// SIMATIC S7-200 project (STEP 7-Micro/WIN), CPU 224 REL 02.01

SYMBOL_TABLE USER1
低压泵延时启动高压        T120
慢驱制动泵启动延时        T110
低压压力正常延时         T109
高压泵工作延时          T108
十分钟停高压泵          T105
运行信号延时           T104
延时停低压泵           T103
再次启高压后停高压        T102
巡检议超温延时          T101
主电机加热            Q5.5
机旁控制指示           Q4.7
机旁反转慢驱指示         Q4.6
机旁正转指示           Q4.5
机旁润滑指示           Q4.4
稀油站出油口温度高        Q4.2
稀油站油位异常          Q4.1
稀油站过滤器故障         Q4.0
稀油站高压油压低         Q3.3
稀油站低压油压低         Q3.2
润滑站油位异常          Q3.1
润滑站油压异常          Q3.0
停止干油泵            Q2.6
系统启动             Q2.5
油站备妥指示           Q2.4
干油泵工作            Q2.3
综合故障输出           Q2.2
停主机信号            Q2.1
油站备妥输出           Q2.0
慢驱油泵工作           Q1.0
慢驱反转             Q0.7
慢驱正转             Q0.6
六泵工作             Q0.5
五泵工作             Q0.4
四号低压泵工作          Q0.3
三号低压泵工作          Q0.2
二泵高压泵工作          Q0.1
一泵高压泵工作          Q0.0
主机停后停干油泵中继       M10.4
慢驱主电机启动前保护       M10.1
慢驱主电机启动后保护       M10.0
停主机中继            M3.3
四号低压泵备用          M3.2
三号低压泵备用          M3.1
总起条件不满足          M3.0
五号润滑泵备用          M2.6
六号润滑泵备用          M2.5
首选手动控制           M2.3
首选自动控制           M2.2
首选机旁控制           M2.1
总起条件             M2.0
急停后再次启高压         M1.5
超温故障停车           M1.6
主机运行记忆           M1.4
主机运行前停车          M1.3     // 主机运行前的停车
高压泵工作            M1.0
启动高压泵            M0.7
低压泵工作            M0.5
手动控制中继           M0.1
内部零电压保护          M0.0
润滑站油温高           I5.7
润滑站油位低           I5.6
润滑站油位高           I5.5
机旁反转慢驱           I5.4
机旁正转慢驱           I5.3
机旁起停润滑           I5.2
机旁启动低压泵          I5.1
机旁起停高压泵          I5.0
润滑油压低            I4.7
润滑压力正常           I4.6
润滑站油压高           I4.5
主机运行             I4.4
低压高              I4.3
稀油站低压低           I4.2
油箱温度低            I4.1
油箱油温高            I4.0
油箱油位低            I3.7
油箱油位高            I3.6
出口油温低            I3.5
出口油温高            I3.4
高低压油站过滤器故障       I3.3
二号高压泵压力低         I3.2
一号高压泵压力低         I3.1
巡检仪超温输入          I3.0
主辅离合器            I2.7     // 开主机为常开
慢驱保护             I2.6
六号泵保护            I2.5
五号泵保护            I2.4
四号泵保护            I2.3
三号泵保护            I2.2
二号泵保护            I2.1
一号泵保护            I2.0
油流控制             I1.5
润滑泵起停            I1.4
低压泵起停            I1.3
高压泵起停            I1.2
润滑泵选择            I1.1
主电机加热温度上限        I0.7
低压泵选择            I1.0
手动加热             I0.6
反转慢驱             I0.5
正转慢驱             I0.4
自动控制             I0.3
机旁控制             I0.2
总起动              I0.1
急停               I0.0     // 主机、机旁、本柜
END_SYMBOL_TABLE

ORGANIZATION_BLOCK 攀枝花紫东钛综合柜程序:OB1
TITLE=【攀枝花矿业公司的空气扫风磨机的自动化控制系统】
// 系统启动前，会检查多项条件，例如油流控制传感器必须正常、主机运行传感器必须未运行、慢驱主电机启动后保护必须未触发，只有这些条件都满足时，总起条件才会置位，允许系统进入运行状态。
// 运行时，系统根据选定的模式和传感器反馈，驱动多个设备。例如，在自动模式下，若油流控制传感器正常且油箱油位低传感器未触发，系统会根据低压泵选择开关的状态，启动三号低压泵工作或四号低压泵工作，但前提是三号泵保护传感器和四号泵保护传感器必须正常，否则泵不会运行。类似地，五号润滑泵工作和六号润滑泵工作的启动需要润滑泵起停按钮或机旁起停润滑按钮的信号，且润滑站油位低传感器未触发，五号泵保护传感器和六号泵保护传感器正常时才能运行。一号高压泵工作和二号高压泵工作则在启动高压泵置位后启动，但需确保一号泵保护传感器和二号泵保护传感器正常。高压泵运行时，若一号高压泵压力低传感器或二号高压泵压力低传感器触发，系统会停止相应的高压泵。
// 系统在启动时检查油站的运行状态。当所有泵运行正常，一号高压泵压力低传感器和二号高压泵压力低传感器未触发，慢驱正转和慢驱反转未运行，主辅离合器传感器正常，且压力参数（如润滑油压低传感器、低压高传感器）和温度参数（如出口油温高传感器、出口油温低传感器）在正常范围内时，油站备妥指示和油站备妥输出才会置位，表示油站准备就绪。油站备妥后，若润滑油压低传感器触发，系统会取消油站备妥指示。若出口油温高传感器触发或手动加热启用，系统启动加热器控制调整温度，确保温度适宜。若油箱温度低触发且油箱油位低未触发，系统可启动加热器。
// 慢驱控制通过正转慢驱按钮、反转慢驱按钮、机旁正转慢驱按钮或机旁反转慢驱按钮操作，启动慢驱油泵工作并控制慢驱正转或慢驱反转。慢驱电机启动时需慢驱保护传感器正常。慢驱运行时，若慢驱保护传感器异常，系统会停止慢驱。干油泵工作则在机旁起停高压泵按钮按下或慢驱运行时启动，提供额外润滑。
// 系统还具备完善的故障保护机制。当润滑站油压异常、润滑站油位异常、稀油站低压油压低、稀油站高压油压低、稀油站过滤器故障、稀油站油位异常、稀油站出油口温度高或慢驱主电机启动前保护等任一异常发生时，综合故障输出会触发，提示操作员检查设备。同时，内部零电压保护只有在延时停低压泵未到时且主机运行前停车未触发时保持置位，确保系统稳定运行。若需要停止主机，停主机信号会在必要时发出。
// 
BEGIN
Network 1 // Network Title
// Network Comment
LD     总起动:I0.1
LDN    高压泵起停:I1.2
AN     低压泵起停:I1.3
AN     润滑泵起停:I1.4
A      手动控制中继:M0.1
LDN    机旁起停润滑:I5.2
AN     油流控制:I1.5
AN     主机运行:I4.4
A      机旁控制:I0.2
OLD
O      自动控制:I0.3
ALD
AN     慢驱主电机启动后保护:M10.0
AN     反转慢驱:I0.5
AN     机旁正转慢驱:I5.3
AN     机旁反转慢驱:I5.4
AN     正转慢驱:I0.4
AN     机旁起停高压泵:I5.0
A      急停:I0.0
=      总起条件:M2.0
Network 2
LD     SM0.0
LD     总起条件:M2.0
O      内部零电压保护:M0.0
ALD
AN     延时停低压泵:T103
AN     主机运行前停车:M1.3
=      内部零电压保护:M0.0
Network 3
LD     SM0.0
LPS
AN     机旁控制:I0.2
AN     自动控制:I0.3
=      手动控制中继:M0.1
LPP
LD     三号低压泵工作:Q0.2
O      五泵工作:Q0.4
O      六泵工作:Q0.5
O      四号低压泵工作:Q0.3
ALD
LPS
LD     机旁控制:I0.2
O      首选机旁控制:M2.1
ALD
AN     首选自动控制:M2.2
AN     首选手动控制:M2.3
=      首选机旁控制:M2.1
LRD
LD     自动控制:I0.3
O      首选自动控制:M2.2
ALD
AN     首选机旁控制:M2.1
AN     首选手动控制:M2.3
=      首选自动控制:M2.2
LPP
LD     手动控制中继:M0.1
O      首选手动控制:M2.3
ALD
AN     首选机旁控制:M2.1
AN     首选自动控制:M2.2
=      首选手动控制:M2.3
Network 4
LDN    稀油站低压低:I4.2
TON    低压压力正常延时:T109, +20
Network 5
LDN    首选机旁控制:M2.1
AN     首选自动控制:M2.2
A      低压泵起停:I1.3
LD     手动控制中继:M0.1
O      三号低压泵工作:Q0.2
O      四号低压泵工作:Q0.3
ALD
LDN    首选自动控制:M2.2
AN     首选手动控制:M2.3
A      油流控制:I1.5
LD     机旁控制:I0.2
O      四号低压泵工作:Q0.3
O      三号低压泵工作:Q0.2
ALD
OLD
LD     自动控制:I0.3
O      四号低压泵工作:Q0.3
O      三号低压泵工作:Q0.2
AN     首选机旁控制:M2.1
AN     首选手动控制:M2.3
OLD
AN     延时停低压泵:T103
AN     油箱油位低:I3.7
A      内部零电压保护:M0.0
LPS
LD     三号低压泵备用:M3.1
ON     低压泵选择:I1.0
ALD
LPS
A      三号泵保护:I2.2
=      三号低压泵工作:Q0.2
LPP
AN     低压压力正常延时:T109
AN     低压高:I4.3
=      四号低压泵备用:M3.2
LPP
LD     四号低压泵备用:M3.2
O      低压泵选择:I1.0
ALD
LPS
A      四号泵保护:I2.3
=      四号低压泵工作:Q0.3
LPP
AN     低压压力正常延时:T109
AN     低压高:I4.3
=      三号低压泵备用:M3.1
Network 6
LD     三号低压泵工作:Q0.2
O      四号低压泵工作:Q0.3
=      低压泵工作:M0.5
TON    低压泵延时启动高压:T120, +20
Network 7
LDN    首选手动控制:M2.3
AN     首选自动控制:M2.2
A      机旁起停润滑:I5.2
LD     机旁控制:I0.2
O      五泵工作:Q0.4
ALD
LDN    首选自动控制:M2.2
AN     首选机旁控制:M2.1
A      润滑泵起停:I1.4
LD     手动控制中继:M0.1
O      五泵工作:Q0.4
ALD
OLD
LD     自动控制:I0.3
O      五泵工作:Q0.4
O      六泵工作:Q0.5
AN     首选机旁控制:M2.1
AN     首选手动控制:M2.3
OLD
AN     润滑站油位低:I5.6
AN     延时停低压泵:T103
A      内部零电压保护:M0.0
AN     润滑站油压高:I4.5
LPS
LDN    润滑泵选择:I1.1
O      五号润滑泵备用:M2.6
ALD
LPS
A      五号泵保护:I2.4
=      五泵工作:Q0.4
LPP
A      润滑油压低:I4.7
=      六号润滑泵备用:M2.5
LPP
LD     润滑泵选择:I1.1
O      六号润滑泵备用:M2.5
ALD
LPS
A      六号泵保护:I2.5
=      六泵工作:Q0.5
LPP
A      润滑油压低:I4.7
=      五号润滑泵备用:M2.6
Network 8
LDN    首选自动控制:M2.2
A      高压泵起停:I1.2
AN     首选机旁控制:M2.1
LD     手动控制中继:M0.1
O      启动高压泵:M0.7
ALD
LDN    首选自动控制:M2.2
A      主机运行:I4.4
AN     首选手动控制:M2.3
LD     机旁控制:I0.2
O      启动高压泵:M0.7
ALD
OLD
LD     自动控制:I0.3
O      启动高压泵:M0.7
LD     五泵工作:Q0.4
O      六泵工作:Q0.5
ALD
AN     首选手动控制:M2.3
AN     首选机旁控制:M2.1
A      低压压力正常延时:T109
A      低压泵延时启动高压:T120
AN     润滑压力正常:I4.6
A      低压泵工作:M0.5
OLD
=      启动高压泵:M0.7
Network 9
LDN    十分钟停高压泵:T105
O      急停后再次启高压:M1.5
A      内部零电压保护:M0.0
A      启动高压泵:M0.7
AN     再次启高压后停高压:T102
LPS
A      一号泵保护:I2.0
=      一泵高压泵工作:Q0.0
LPP
A      二号泵保护:I2.1
=      二泵高压泵工作:Q0.1
Network 10
LD     机旁起停高压泵:I5.0
TON    十分钟停高压泵:T105, +18000
Network 11
LD     一泵高压泵工作:Q0.0
O      二泵高压泵工作:Q0.1
=      高压泵工作:M1.0
Network 12
LDN    一号高压泵压力低:I3.1
A      一泵高压泵工作:Q0.0
LD     二泵高压泵工作:Q0.1
AN     二号高压泵压力低:I3.2
OLD
O      机旁起停高压泵:I5.0
LD     五泵工作:Q0.4
O      六泵工作:Q0.5
ALD
LD     三号低压泵工作:Q0.2
O      四号低压泵工作:Q0.3
ALD
AN     慢驱正转:Q0.6
AN     慢驱反转:Q0.7
AN     主辅离合器:I2.7
LDN    一号高压泵压力低:I3.1
A      一泵高压泵工作:Q0.0
LD     二泵高压泵工作:Q0.1
AN     二号高压泵压力低:I3.2
OLD
LD     五泵工作:Q0.4
O      六泵工作:Q0.5
ALD
LD     三号低压泵工作:Q0.2
O      四号低压泵工作:Q0.3
ALD
AN     机旁起停高压泵:I5.0
A      主辅离合器:I2.7
OLD
A      低压压力正常延时:T109
AN     润滑油压低:I4.7
AN     低压高:I4.3
AN     润滑站油压高:I4.5
AN     综合故障输出:Q2.2
TON    T111, +2
Network 13
LD     T111
=      油站备妥指示:Q2.4
A      内部零电压保护:M0.0
=      油站备妥输出:Q2.0
Network 14
LD     正转慢驱:I0.4
O      反转慢驱:I0.5
O      机旁正转慢驱:I5.3
O      机旁反转慢驱:I5.4
O      慢驱油泵工作:Q1.0
AN     机旁起停高压泵:I5.0
A      内部零电压保护:M0.0
A      主辅离合器:I2.7
A      慢驱保护:I2.6
=      慢驱油泵工作:Q1.0
Network 15
LD     慢驱油泵工作:Q1.0
TON    慢驱制动泵启动延时:T110, +10
Network 16
LD     机旁控制:I0.2
O      慢驱正转:Q0.6
AN     首选手动控制:M2.3
A      机旁正转慢驱:I5.3
LD     手动控制中继:M0.1
O      慢驱正转:Q0.6
LDN    机旁正转慢驱:I5.3
A      正转慢驱:I0.4
LDN    正转慢驱:I0.4
A      机旁正转慢驱:I5.3
OLD
ALD
AN     首选机旁控制:M2.1
OLD
A      慢驱制动泵启动延时:T110
AN     首选自动控制:M2.2
AN     慢驱反转:Q0.7
=      慢驱正转:Q0.6
Network 17
LD     机旁控制:I0.2
O      慢驱反转:Q0.7
AN     首选手动控制:M2.3
A      机旁反转慢驱:I5.4
LD     手动控制中继:M0.1
O      慢驱反转:Q0.7
LDN    机旁反转慢驱:I5.4
A      反转慢驱:I0.5
LDN    反转慢驱:I0.5
A      机旁反转慢驱:I5.4
OLD
ALD
AN     首选机旁控制:M2.1
OLD
AN     首选自动控制:M2.2
A      慢驱制动泵启动延时:T110
AN     慢驱正转:Q0.6
=      慢驱反转:Q0.7
Network 18
LD     机旁起停高压泵:I5.0
O      慢驱正转:Q0.6
O      慢驱反转:Q0.7
TON    运行信号延时:T104, +10
A      运行信号延时:T104
A      内部零电压保护:M0.0
AN     停止干油泵:Q2.6
=      干油泵工作:Q2.3
Network 19
LD     干油泵工作:Q2.3
A      内部零电压保护:M0.0
=      系统启动:Q2.5
Network 20
LD     SM0.0
LPS
AN     机旁启动低压泵:I5.1
TON    T127, +100
LRD
A      油箱温度低:I4.1
TON    T128, +100
LRD
A      出口油温低:I3.5
TON    T129, +100
LPP
LD     手动加热:I0.6
O      T128
O      T129
ALD
A      T127
AN     机旁启动低压泵:I5.1
A      内部零电压保护:M0.0
AN     油箱油位低:I3.7
=      Q5.4
Network 21
LD     机旁控制:I0.2
A      主电机加热温度上限:I0.7
A      内部零电压保护:M0.0
=      主电机加热:Q5.5
Network 22
LD     SM0.0
LPS
LD     润滑站油压高:I4.5
A      内部零电压保护:M0.0
LD     T151
A      M3.5
OLD
ALD
=      润滑站油压异常:Q3.0
LPP
A      低压高:I4.3
TOF    T151, +100
A      内部零电压保护:M0.0
AN     总起动:I0.1
=      M3.5
Network 23
LD     润滑站油位低:I5.6
O      润滑站油位高:I5.5
A      内部零电压保护:M0.0
=      润滑站油位异常:Q3.1
Network 24
LD     稀油站低压低:I4.2
A      低压泵工作:M0.5
A      内部零电压保护:M0.0
=      稀油站低压油压低:Q3.2
Network 25
LD     高压泵工作:M1.0
TON    高压泵工作延时:T108, +100
Network 26
LD     一泵高压泵工作:Q0.0
A      一号高压泵压力低:I3.1
LD     二泵高压泵工作:Q0.1
A      二号高压泵压力低:I3.2
OLD
A      高压泵工作延时:T108
A      内部零电压保护:M0.0
=      稀油站高压油压低:Q3.3
Network 27
LD     高低压油站过滤器故障:I3.3
A      内部零电压保护:M0.0
=      稀油站过滤器故障:Q4.0
Network 28
LD     油箱油位低:I3.7
O      油箱油位高:I3.6
A      内部零电压保护:M0.0
=      稀油站油位异常:Q4.1
Network 29
LD     出口油温高:I3.4
A      内部零电压保护:M0.0
=      稀油站出油口温度高:Q4.2
Network 30
LD     五泵工作:Q0.4
O      六泵工作:Q0.5
LD     机旁控制:I0.2
O      机旁润滑指示:Q4.4
ALD
A      内部零电压保护:M0.0
AN     首选自动控制:M2.2
AN     首选手动控制:M2.3
=      机旁润滑指示:Q4.4
Network 31
LD     机旁正转慢驱:I5.3
A      内部零电压保护:M0.0
A      慢驱正转:Q0.6
=      机旁正转指示:Q4.5
Network 32
LD     机旁反转慢驱:I5.4
A      内部零电压保护:M0.0
A      慢驱反转:Q0.7
=      机旁反转慢驱指示:Q4.6
Network 33
LD     机旁控制:I0.2
O      机旁控制指示:Q4.7
AN     首选自动控制:M2.2
A      内部零电压保护:M0.0
AN     首选手动控制:M2.3
=      机旁控制指示:Q4.7
Network 34
LD     总起动:I0.1
AN     总起条件:M2.0
AN     内部零电压保护:M0.0
=      总起条件不满足:M3.0
Network 35
LD     润滑站油压异常:Q3.0
O      润滑站油位异常:Q3.1
O      稀油站低压油压低:Q3.2
O      稀油站高压油压低:Q3.3
O      稀油站过滤器故障:Q4.0
O      稀油站油位异常:Q4.1
O      稀油站出油口温度高:Q4.2
O      慢驱主电机启动前保护:M10.1
O      慢驱主电机启动后保护:M10.0
O      低压高:I4.3
A      内部零电压保护:M0.0
O      总起条件不满足:M3.0
LPS
AN     T125
=      综合故障输出:Q2.2
LPP
TON    T125, +10
Network 36
LD     巡检仪超温输入:I3.0
TON    巡检议超温延时:T101, +300
Network 37
LD     巡检议超温延时:T101
A      内部零电压保护:M0.0
=      超温故障停车:M1.6
Network 38
LD     机旁起停高压泵:I5.0
O      主机运行记忆:M1.4
LPS
A      内部零电压保护:M0.0
TON    T122, +300
LRD
A      T122
=      主机运行记忆:M1.4
LPP
AN     机旁起停高压泵:I5.0
=      主机停后停干油泵中继:M10.4
Network 39
LDN    急停:I0.0
O      慢驱主电机启动前保护:M10.1
LPS
A      主机运行记忆:M1.4
LPS
AN     机旁起停高压泵:I5.0
TON    再次启高压后停高压:T102, +9000
LRD
=      急停后再次启高压:M1.5
LPP
=      停主机中继:M3.3
LPP
AN     主机运行记忆:M1.4
=      主机运行前停车:M1.3
Network 40
LD     SM0.0
LD     机旁起停高压泵:I5.0
O      慢驱正转:Q0.6
O      慢驱反转:Q0.7
ALD
LPS
LD     一泵高压泵工作:Q0.0
O      M8.0
ALD
=      M8.0
LRD
LD     二泵高压泵工作:Q0.1
O      M8.1
ALD
=      M8.1
LRD
LD     三号低压泵工作:Q0.2
O      M8.2
ALD
=      M8.2
LRD
LD     四号低压泵工作:Q0.3
O      M8.3
ALD
=      M8.3
LRD
LD     五泵工作:Q0.4
O      M8.4
ALD
=      M8.4
LPP
LD     六泵工作:Q0.5
O      M8.5
ALD
=      M8.5
Network 41
LD     SM0.0
LPS
AN     一号泵保护:I2.0
LPS
A      M8.0
=      M4.0
LPP
AN     内部零电压保护:M0.0
=      M4.1
LRD
AN     二号泵保护:I2.1
LPS
A      M8.1
=      M4.2
LPP
AN     内部零电压保护:M0.0
=      M4.3
LRD
AN     三号泵保护:I2.2
LPS
A      M8.2
=      M4.4
LPP
AN     内部零电压保护:M0.0
=      M4.5
LRD
AN     四号泵保护:I2.3
LPS
A      M8.3
=      M4.6
LPP
AN     内部零电压保护:M0.0
=      M4.7
LRD
AN     五号泵保护:I2.4
LPS
A      M8.4
=      M5.0
LPP
AN     内部零电压保护:M0.0
=      M5.1
LRD
AN     六号泵保护:I2.5
LPS
A      M8.5
=      M5.2
LPP
AN     内部零电压保护:M0.0
=      M5.3
LRD
LD     M4.0
O      M4.2
O      M4.4
O      M4.6
O      M5.0
O      M5.2
ON     慢驱保护:I2.6
ALD
=      慢驱主电机启动前保护:M10.1
LPP
LD     M4.1
O      M4.3
O      M4.5
O      M4.7
O      M5.1
O      M5.3
ON     慢驱保护:I2.6
ALD
=      慢驱主电机启动后保护:M10.0
Network 42
LD     停主机中继:M3.3
O      主辅离合器:I2.7
O      超温故障停车:M1.6
O      润滑站油位异常:Q3.1
O      慢驱主电机启动后保护:M10.0
O      稀油站油位异常:Q4.1
O      主机停后停干油泵中继:M10.4
AN     总起动:I0.1
=      停主机信号:Q2.1
Network 43
LDN    机旁起停高压泵:I5.0
AN     干油泵工作:Q2.3
LDN    慢驱反转:Q0.7
AN     首选自动控制:M2.2
AN     慢驱正转:Q0.6
OLD
AN     一泵高压泵工作:Q0.0
AN     二泵高压泵工作:Q0.1
A      急停后再次启高压:M1.5
A      再次启高压后停高压:T102
TON    延时停低压泵:T103, +60
Network 44
LD     停主机中继:M3.3
O      超温故障停车:M1.6
O      润滑站油位异常:Q3.1
O      慢驱主电机启动后保护:M10.0
O      稀油站油位异常:Q4.1
O      主机停后停干油泵中继:M10.4
O      主机运行前停车:M1.3
LDN    机旁起停高压泵:I5.0
AN     慢驱正转:Q0.6
AN     慢驱反转:Q0.7
OLD
LPS
LD     内部零电压保护:M0.0
O      主机运行前停车:M1.3
ALD
AN     T117
AN     总起动:I0.1
=      停止干油泵:Q2.6
LPP
TON    T117, +100
END_ORGANIZATION_BLOCK

// SBR1: protected block, not included

// INT1: protected block, not included

// (further data pages could not be read)
